FUNCTION_BLOCK controller
  (* Standard: 61499-2 *)
  (* Version 0.1, 2015-00-13, Th?o, PC_THEO *)
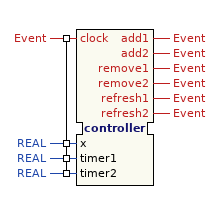
  EVENT_INPUT
    clock WITH x, timer1, timer2;
  END_EVENT
  EVENT_OUTPUT
    add1;
    add2;
    remove1;
    remove2;
    refresh1;
    refresh2;
  END_EVENT
  VAR_INPUT
    x : REAL;
    timer1 : REAL;
    timer2 : REAL;
  END_VAR
  VAR
    y1 : REAL;
    y2 : REAL;
    c : REAL;
  END_VAR
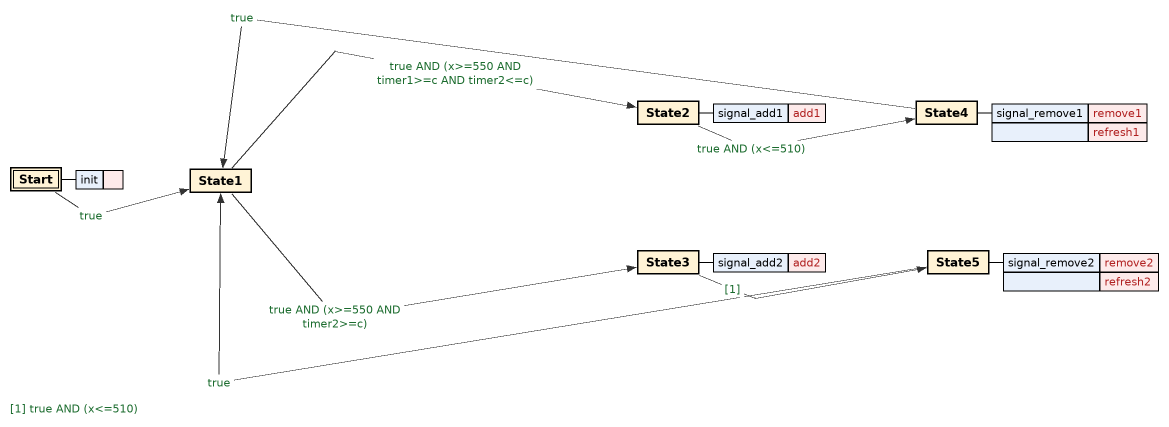
  EC_STATES
    Start : init;
    State1;
    State2 : signal_add1 -> add1;
    State3 : signal_add2 -> add2;
    State4 : signal_remove1 -> remove1, -> refresh1;
    State5 : signal_remove2 -> remove2, -> refresh2;
  END_STATES
  EC_TRANSITIONS
    Start TO State1 := true;
    State1 TO State3 := true AND (x>=550 AND timer2>=c);
    State1 TO State2 := true AND (x>=550 AND timer1>=c AND timer2<=c);
    State2 TO State4 := true AND (x<=510);
    State3 TO State5 := true AND (x<=510);
    State4 TO State1 := true;
    State5 TO State1 := true;
  END_TRANSITIONS
  ALGORITHM init IN C:
me->x=510;
me->c=20;
  END_ALGORITHM
  ALGORITHM signal_add2 IN C:
printf("Send signal: add2, Temperature : %f\n",me->x);
  END_ALGORITHM
  ALGORITHM signal_add1 IN C:
printf("Send signal: add1, Temperature : %f\n",me->x);
  END_ALGORITHM
  ALGORITHM signal_remove1 IN C:
printf("Send signal: remove1, Temperature : %f\n",me->x);
  END_ALGORITHM
  ALGORITHM signal_remove2 IN C:
printf("Send signal: remove2, Temperature : %f\n",me->x);
  END_ALGORITHM
END_FUNCTION_BLOCK
